(* PLC project Unnamed, Unknown Unnamed 1 *)
(* stored: creationDateTime 2022-10-30T21:25:48, modificationDateTime 2022-11-20T19:39:50 *)

FUNCTION_BLOCK TC006
  VAR_INPUT
    i1 : BOOL;
    i2 : BOOL;
    i3 : BOOL;
    i4 : BOOL;
  END_VAR
  VAR_OUTPUT
    o1 : BOOL;
    o2 : BOOL;
    o3 : BOOL;
    o4 : BOOL;
    o5 : BOOL;
  END_VAR
  VAR
    l1 : BOOL;
    l2 : TIME := T#5s;
    l3 : TIME := T#2s;
    l4 : BOOL;
    TON0 : TON;
    TOF0 : TOF;
  END_VAR
  VAR  (* added by the conversion: wires and edge detectors of the diagram *)
    _AND1_OUT : BOOL;
  END_VAR

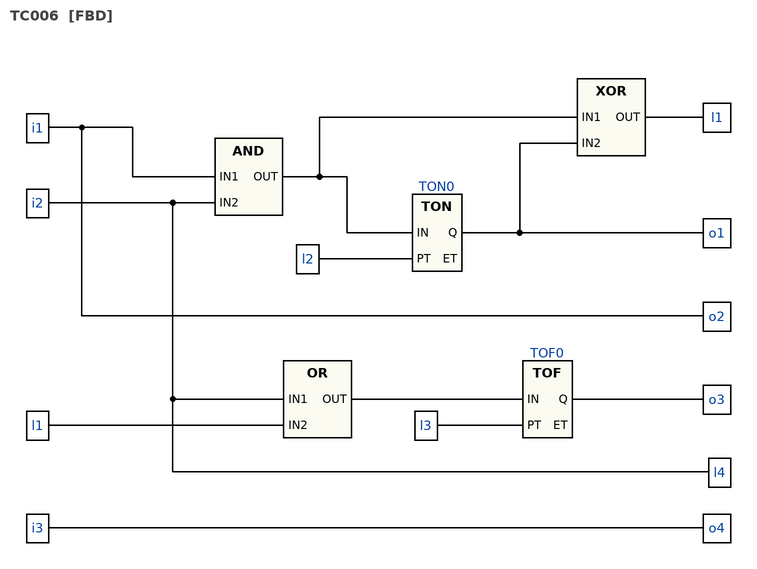
(* FBD diagram, written out as Structured Text *)
_AND1_OUT := i1 AND i2;
TON0(IN := _AND1_OUT, PT := l2);
l1 := _AND1_OUT XOR TON0.Q;
o1 := TON0.Q;
o2 := i1;
TOF0(IN := i2 OR l1, PT := l3);
o3 := TOF0.Q;
l4 := i2;
o4 := i3;
END_FUNCTION_BLOCK

CONFIGURATION config
  RESOURCE resource1 ON PLC
  END_RESOURCE
END_CONFIGURATION
